Universal Robots PolyScope program: xml_rpc_sample.urp

Program xml_rpc_sample (installation=default directory=/home/ur/ursim-current/programs createdIn=5.11.0.108249 lastSavedIn=5.6.0.90886 robotSerialNumber=20195699999)
Calibrated DH parameters: a=[0, -0.4784, -0.36, 0, 0, 0]; d=[0.1807, 0, 0, 0.17415, 0.11985, 0.11655]; alpha=[1.570796, 0, 0, 1.570796, -1.570796, 0]; deltaTheta=[0, 0, 0, 0, 0, 0]
InitVariablesNode
Robot Program (runOnlyOnce=true)
  'Connection to the remote PC (change the IP to match the IP of the PC running the SDK)'
  rpc := rpc_factory("xmlrpc","http://192.168.0.10:50000")
  'Remote call the method get_answer with arguments and wait for answer'
  answer1 := rpc.get_answer("Hello",  True ,  False , 12, 12.2, p[100,100,120,0.1,0,0], [12, 1.2,123])
  answer2 := rpc.rpc.GetPose()
  answer3 := rpc.HowAreYou("Alfred")
  answer4 := rpc.SumFirstArray([1,3.5,-2])
  answer5 := rpc.SumMyArguments(1,3.5,-2)
  'Simple call to the method getPose with no arguments and no returned value'
  Script: rpc.nothingReturned()
